// TIA Portal V17 export
// export: Created 2025-01-08T13:55:34.3139256Z, ExportSetting WithDefaults, DisplayName Totally Integrated Automation Portal, DisplayVersion V17, DisplayName TIA Portal Openness, DisplayVersion V17, DisplayName TIA Portal Version Control Interface, DisplayVersion V17, DisplayName SINAMICS Startdrive Advanced, DisplayVersion V17 Update2, DisplayName SINAMICS Startdrive G130, G150, S120, S150, SINAMICS MV, S210, DisplayVersion V17 Update2, DisplayName SINAMICS Startdrive G110M, G120, G120C, G120D, G120P, G115D, DisplayVersion V17 Update2, DisplayName STEP 7 Professional, DisplayVersion V17, DisplayName STEP 7 Safety, DisplayVersion V17, DisplayName WinCC Advanced, DisplayVersion V17
DATA_BLOCK "DB - Events_To_PC"   // DB26
{ S7_Optimized_Access := 'FALSE' }
VERSION : 0.1
// stored: AutoNumber true, DBAccessibleFromOPCUA true, DBAccessibleFromWebserver true, IsOnlyStoredInLoadMemory false, IsWriteProtectedInAS false
   VAR
      ADoorNotClosed : Bool;   // Door to Index Wheel not Closed
      ANoLabelGapFound : Bool;   // Kontrollera etikettladdning vid etikett givare
      ARewinderTimeOut : Bool;   // Kontrollera etikettladdning vid upprullare
      WExternalPause : Bool;   // Machine paused by external machine
      ANoLabel_In_LabelQueue : Bool;   // Ingen Etikett hittad i etikettkö
      AStopInReject : Bool;   // Product stuck in side outfeed
      ACam4_Max_Rejects_Reached : Bool;   // Cam 4 max rejects reached. Check Camera HMI.
      AE_Stop_Not_Ok : Bool;   // Safety circuit not okay. Check emergency buttons and reset.
      ALabelEndOnActiveUnwinder : Bool;   // Etikett slut
      WLabelLowUnwinder1 : Bool;   // Etikett låg avrullare 1
      WLabelLowUnwinder2 : Bool;   // Etikett låg avrullare 2
      ILabelSeamedEvent : Bool;   // Label Seamed
      ACam3_Max_Rejects_Reached : Bool;   // Camera 3 max rejects reached. Check Camera HMI
      AFeed_Label_Drive_Error : Bool;   // Fel på motor till Kö
      ADispense_Label_Drive_Error : Bool;   // Fel på motor till Etikett Dispensering
      ARotate_Product_Drive_Error : Bool;   // Fault with rotate product motor.
      AIndex_Wheel_Drive_Error : Bool;   // Fault with index wheel motor.
      ARewinder_Drive_Error : Bool;   // Fel på motor till Upprullare
      AFindLabelGap_Error : Bool;   // Fel på kommunikation mellan Dispenerings drive och PLC
      AZone2_Conveyor_Error : Bool;   // Fault Zone 2 conveyor motor
      AZone2_Queue_Error : Bool;   // Fault Zone 2 queue motor.
      AZone2_Side_HSM_Move_Error : Bool;   // Fault Zone 2 Label adjust motor.
      ARotation_Error : Bool;   // Fault with product orientation motor. Either left or right.
      AZone2_Side_HSM_Error : Bool;   // Fault Zone 2 side motors labeling.
      AZone1_Conveyor_Error : Bool;   // Fault Zone 1 conveyor motor,
      AZone1_Queue_Error : Bool;   // Fault Zone 1 queue motor.
      AZone1_Side_HSM_Error : Bool;   // Fault Zone 1 side motors labeling.
      ANo_Product_In_Index_Wheel : Bool;   // No Product in Index Wheel.
      AZone1ConveyorFull : Bool;   // Zone 1 Conveyor full of products. Clear products and start machine.
      AZone2ConveyorFull : Bool;   // Zone 2 Conveyor full of products. Clear products and start machine.
      ARewinderFull : Bool;   // Upprullaren är full
      AHSMSideNotOK : Bool;   // HSM Side is not Ready.
      AHSMZon1NotOK : Bool;   // HSM Zone 1 is not Ready.
      AHSMZon2NotOK : Bool;   // HSM Zone 2 is not Ready.
      AMachineStoppedByWatchdog : Bool;   // Machine stopped by lost connection between HMI and PLC.
      IIgnoreExternalPauseActive : Bool;   // Ignore External Pause is activated.
      IJogFunctionActive : Bool;   // Jog function is activated.
      IStandbyFunctionDeactivated : Bool;   // Standby function is deactivated.
      WStanbyIsActive : Bool;   // Standby is active and the machine can start by it self.
      WWarningFromHSM_Side : Bool;   // Warning from Side HSM.
      WWarningFromHSM_Zon1 : Bool;   // Warning from Zone 1 HSM.
      WWarningFromHSM_Zon2 : Bool;   // Warning from Zone 2 HSM.
      ATop_Side_HSM_Move_Error : Bool;   // Fault Zone 1 Label adjust motor.
      IEmptyMachineRunning : Bool;   // Machine will run until there's no more products and stop.
      ALowAirPressure : Bool;   // Low air pressure check air and air pressure.
      ICam1Deactivated : Bool;   // Camera 1 deactivated.
      ICam2Deactivated : Bool;   // Camera 2 deactivated.
      ICam3Deactivated : Bool;   // Camera 3 deactivated.
      ICam4Deactivated : Bool;   // Camera 4 deactivated.
      IHSMSideDeactivated : Bool;   // HSM Side deactivated.
      IHSMZone1Deactivated : Bool;   // HSM Zone 1 deactivated.
      IHSMZone2Deactivated : Bool;   // HSM Zone 2 deactivated.
      WSideRejectFull : Bool;   // Reject låda till banderoll full
      ACam1_Max_Rejects_Reached : Bool;   // Camera 1 max rejects reached. Check Camera HMI.
      ISpeed_1 : Bool;   // Speed 1 selected.
      ISpeed_2 : Bool;   // Speed 2 Selected.
      ISpeed_3 : Bool;   // Speed 3 Selected.
      ISpeed_4 : Bool;   // Speed 4 Selected.
      ISpeed_5 : Bool;   // Speed 5 Selected.
      ABufferConveyorFault : Bool;   // Engine protection tripped on buffer conveyor.
      AAC_NotReady : Bool;   // 4050AC is not ready.
      WAC_Warning : Bool;   // Warning from 4050AC.
      IIndexWheelHoming : Bool;   // Index Wheel homing or waiting for products to start homing.
      APrinterNotReady : Bool;   // Printer is not ready
      IPrinterDeactivated : Bool;   // Printer deactivated
      MachineSpeed : Real := 50.0;
   END_VAR
BEGIN
END_DATA_BLOCK
